(* CoDeSys 2.3.8.1 project: coconuts.pro *)
(* Libraries: C:\Program Files (x86)\Common Files\CAA-Targets\3S\Lib_PLCWinNT\SysLibTime.lib 23.9.04 10:11:36, STANDARD.LIB 4.10.05 11:14:46, IECSFC.LIB 13.4.06 15:51:28, Util.lib 1.6.07 09:40:58, ANALYZATION.LIB 5.10.99 09:05:06, C:\Program Files (x86)\Common Files\CAA-Targets\3S\Lib_PLCWinNT\SysLibFile.lib 23.9.04 10:11:36 *)

(* PLC configuration (modules and I/O channels)
Discrete input 6 bit [ID100] node 0, in %IB0 out %QB0 {Filtrationtime = 10; Filtrationtime = 10; Filtrationtime = 10; Filtrationtime = 10; Filtrationtime = 10; Filtrationtime = 10; Visibility = No; PinCount = 6; WatchDogPeriod = 1000; PollPeriod = 1}
  SW1 AT %IX0.0 [BitInput]
  SW2 AT %IX0.1 [BitInput]
  SW3 AT %IX0.2 [BitInput]
  SW4 AT %IX0.3 [BitInput] kitchen
  SW5 AT %IX0.4 [BitInput]
  SW6 AT %IX0.5 [BitInput] entrance
R1 AT %QX1.0 [BitOutput] water boiler
_R2 AT %QX1.1 [BitOutput]
_R3 AT %QX1.2 [BitOutput] entrance
R4 AT %QX1.3 [BitOutput] electro boiler
Special output [ID104] node 2, in %IB2 out %QB2 {Visibility = No; PinCount = 1}
  BEEPER AT %QX2.0 [BitOutput] Special output
Unifed signal sensor [ID700] node 3, in %IB3 out %QB3 {Type_of_sensor700 = U0_1; measure_interval = 1; ainlow = 0; ainhigh = 30; first_cor_point = 0; first_delta = 0; second_cor_point = 0; second_delta = 0; third_cor_point = 0; third_delta = 0; Visibility = No}
  AT %ID3.0 [FloatInput] Value
  AT %IW3.1 [WordInput] Circular time
  Analog Input [ID107] node 0, in %IB3.0 out %QB3.0
Unifed signal sensor [ID700] node 4, in %IB4 out %QB4 {Type_of_sensor700 = U0_1; measure_interval = 0.5; ainlow = 0; ainhigh = 20; first_cor_point = 0; first_delta = 0; second_cor_point = 0; second_delta = 0; third_cor_point = 0; third_delta = 0; Visibility = No}
  AT %ID4.0 [FloatInput] Value
  AT %IW4.1 [WordInput] Circular time
  Analog Input [ID107] node 0, in %IB4.0 out %QB4.0
Unifed signal sensor [ID700] node 5, in %IB5 out %QB5 {Type_of_sensor700 = U0_1; measure_interval = 0.5; ainlow = 0; ainhigh = 20; first_cor_point = 0; first_delta = 0; second_cor_point = 0; second_delta = 0; third_cor_point = 0; third_delta = 0; Visibility = No}
  AT %ID5.0 [FloatInput] Value
  AT %IW5.1 [WordInput] Circular time
  Analog Input [ID107] node 0, in %IB5.0 out %QB5.0
Unifed signal sensor [ID700] node 6, in %IB6 out %QB6 {Type_of_sensor700 = U0_1; measure_interval = 0.5; ainlow = 0; ainhigh = 20; first_cor_point = 0; first_delta = 0; second_cor_point = 0; second_delta = 0; third_cor_point = 0; third_delta = 0; Visibility = No}
  AT %ID6.0 [FloatInput] Value
  AT %IW6.1 [WordInput] Circular time
  Analog Input [ID107] node 0, in %IB6.0 out %QB6.0
Analog output [ID106] node 7, in %IB7 out %QB7 {DAC_Type = Voltage 0-10 B; Analog_offset_correction = 0; Analog_full_range_correction = 0; SafeValueFloat = 0; Visibility = No}
  AT %QD7.0 [FloatOutput] Value
Analog output [ID106] node 8, in %IB8 out %QB8 {DAC_Type = Voltage 0-10 B; Analog_offset_correction = 0; Analog_full_range_correction = 0; SafeValueFloat = 0; Visibility = No}
  AT %QD8.0 [FloatOutput] Value
ModBus (Master) [MODBUS_MASTER_ID450] node 9, in %IB9 out %QB9 {Visibility = No}
  MODBUS_LAST_ADDR AT %QD9.0 [DWordOutput] Last address
  MODBUS_LAST_ERROR AT %QW9.1 [WordOutput] Last error
  RS-485-1 [COM1_USART] node 0, in %IB9.0 out %QB9.0 {CommunicationSpeed = 9600; Parity = NO PARITY CHECK; BitLength = 8 bits; StopLength = One stop bit; InterfaceType = RS485; FrameOriented = RTU; Timeout = 0; Visibility = No}
  Universal Modbus device [ID2000] node 1, in %IB9.1 out %QB9.1 {ModuleIP = 10:0:0:223; ServiceTimeout = 150; TCPport = 502; NetMode = Serial; ModuleSlaveAddress = 3; RequestType = By poll time; PeriodOfService = 5000; Visibility = Yes; RepeatCounter = 0; ByteSequence = Trace_mode}
    AT %QB9.1.0 [ComChannel] Command (0xff - Start)
temp8 AT %IW9.1.0.0 [WordInput]
temp7 AT %IW9.1.1.0 [WordInput]
temp6 AT %IW9.1.2.0 [WordInput]
temp5 AT %IW9.1.3.0 [WordInput] 2f bedroom
temp4 AT %IW9.1.4.0 [WordInput] bath warm floor
temp3 AT %IW9.1.5.0 [WordInput] coolant
temp2 AT %IW9.1.6.0 [WordInput] living room
temp1 AT %IW9.1.7.0 [WordInput] boiler
Universal Modbus device [ID2000] node 2, in %IB9.2 out %QB9.2 {ModuleIP = 10:0:0:223; ServiceTimeout = 150; TCPport = 502; NetMode = Serial; ModuleSlaveAddress = 7; RequestType = By poll time; PeriodOfService = 5000; Visibility = Yes; RepeatCounter = 0; ByteSequence = Trace_mode}
  AT %QB9.2.0 [ComChannel] Command (0xff - Start)
temp78 AT %IW9.2.0.0 [WordInput] bedroom 2f
temp77 AT %IW9.2.1.0 [WordInput] hall
temp76 AT %IW9.2.2.0 [WordInput]
temp75 AT %IW9.2.3.0 [WordInput]
temp74 AT %IW9.2.4.0 [WordInput]
temp73 AT %IW9.2.5.0 [WordInput]
temp72 AT %IW9.2.6.0 [WordInput]
temp71 AT %IW9.2.7.0 [WordInput]
Universal Modbus device [ID2000] node 3, in %IB9.3 out %QB9.3 {ModuleIP = 10:0:0:223; ServiceTimeout = 150; TCPport = 502; NetMode = Serial; ModuleSlaveAddress = 2; RequestType = By poll time; PeriodOfService = 100; Visibility = Yes; RepeatCounter = 0; ByteSequence = Trace_mode}
  AT %QB9.3.0 [ComChannel] Command (0xff - Start)
AT %QB9.3.0.0 [ByteOutput]
Universal Modbus device [ID2000] node 4, in %IB9.4 out %QB9.4 {ModuleIP = 10:0:0:223; ServiceTimeout = 150; TCPport = 502; NetMode = Serial; ModuleSlaveAddress = 6; RequestType = By poll time; PeriodOfService = 100; Visibility = No; RepeatCounter = 0; ByteSequence = Trace_mode}
  AT %QB9.4.0 [ComChannel] Command (0xff - Start)
  8 bit input module [ID2001] node 0, in %IB9.4.0 out %QB9.4.0 {ModbusAddress = 0; Command_read_byte = Read inputs status  (0x02); Visibility = No}
    AT %IB9.4.0.0 [ByteInput]
AT %QB9.4.1.0 [ByteOutput]
AT %QB9.5.0 [ComChannel] Command (0xff - Start)
AT %QB9.5.0.0 [ByteOutput]
AT %IB9.5.1.0 [ByteInput]
Universal Modbus device [ID2000] node 6, in %IB9.6 out %QB9.6 {ModuleIP = 10:0:0:223; ServiceTimeout = 150; TCPport = 502; NetMode = Serial; ModuleSlaveAddress = 11; RequestType = By poll time; PeriodOfService = 20; Visibility = No; RepeatCounter = 0; ByteSequence = Trace_mode}
  AT %QB9.6.0 [ComChannel] Command (0xff - Start)
current AT %ID9.6.0.0 [FloatInput]
power AT %ID9.6.1.0 [FloatInput]
voltage AT %ID9.6.2.0 [FloatInput]
total_energy AT %ID9.6.3.0 [FloatInput]
Modbus [MODBUS_ID302] node 0, in %IB10.0 out %QB10.0
  TCP [TCP_ID221] node 0, in %IB10.0.0 out %QB10.0.0 {RemotePort = 502; Visibility = No}
REG0_LIGHTS16 AT %QW10.1.0 [WordOutput] reg0
REG1_PLC_FLAGS AT %QW10.2.0 [WordOutput] reg1
REG2_BOILERS AT %QW10.3.0 [WordOutput] reg2
REG3_PUMPS AT %QW10.4.0 [WordOutput] reg3
REG4_BATH_FAN_MODE AT %QW10.5.0 [WordOutput] reg4
REG5 AT %QW10.6.0 [WordOutput] reg5
REG6_LIVING_ROOM_TERMOSTAT_DESIRED AT %QW10.7.0 [WordOutput] reg6
REG7_HALL_TERMOSTAT_DESIRED AT %QW10.8.0 [WordOutput] reg7
REG8_2F_BEDROOM_TERMOSTAT_DESIRED AT %QW10.9.0 [WordOutput] reg8
REG9 AT %QW10.10.0 [WordOutput] reg9
REG10_TEMP1 AT %QW10.11.0 [WordOutput] reg10
REG11_TEMP2 AT %QW10.12.0 [WordOutput] reg11
REG12_TEMP3 AT %QW10.13.0 [WordOutput] reg12
REG13_TEMP4 AT %QW10.14.0 [WordOutput] reg13
REG14_TEMP5 AT %QW10.15.0 [WordOutput] reg14
REG15_TEMP6 AT %QW10.16.0 [WordOutput] reg15
REG16_TEMP7 AT %QW10.17.0 [WordOutput] reg16
REG17_TEMP8 AT %QW10.18.0 [WordOutput] reg17
REG18 AT %QW10.19.0 [WordOutput] reg18
REG19 AT %QW10.20.0 [WordOutput] reg19
REG20 AT %QW10.21.0 [WordOutput] reg20
REG21_POWER AT %QW10.22.0 [WordOutput]
REG22_VOLTAGE AT %QW10.23.0 [WordOutput]
REG23_TOTAL_ENERGY AT %QW10.24.0 [WordOutput]
REG24_TIME AT %QW10.25.0 [WordOutput]
ID4002 byteIB
%QB
%MB
%MREG25_MODBUS_ERRORS AT %QW10.26.0 [WordOutput]
REG26_BOILER_DESIRED_TEMP AT %QW10.27.0 [WordOutput]
REG27_BOILER_CUR_TEMP AT %QW10.28.0 [WordOutput]
REG28_BOILER_MODE AT %QW10.29.0 [WordOutput]
REG29_TEMP71 AT %QW10.30.0 [WordOutput]
REG30_TEMP72 AT %QW10.31.0 [WordOutput]
REG31_TEMP73 AT %QW10.32.0 [WordOutput]
REG32_TEMP74 AT %QW10.33.0 [WordOutput]
REG33_TEMP75 AT %QW10.34.0 [WordOutput]
REG34_TEMP76 AT %QW10.35.0 [WordOutput]
REG35_TEMP77 AT %QW10.36.0 [WordOutput]
REG36_TEMP78 AT %QW10.37.0 [WordOutput]
*)

(* Global variable list: Global_Variables *)
VAR_GLOBAL
	RO_POWER_NIGHT_MODE: BOOL;
	RO_POWER_SAFE_MODE:BOOL;

	WATER_BOILER_STATE:BOOL;
	RO_WATER_BOILER_VALVE_STATE:BOOL;

	RO_WARM_FLOOR_PUMP_STATE:BOOL;

	RO_LIVINGROOM_TERMOSTAT_STATE:BOOL;
	RO_BEDROOM_2F_TERMOSTAT_STATE:BOOL;

	RO_BEDROOM_2F_VALVE_STATE:BOOL;
	RO_HALL_VALVE_STATE:BOOL;

	TOWEL_HEATER_SW:switch;
	BATH_LIGHT_SW:switch;

	RO_BATH_FAN_STATE:BOOL;
END_VAR

VAR_GLOBAL CONSTANT
	MIN_COOLANT_TEMP: WORD := 300;
	MAX_COOLANT_TEMP: WORD := 600;
END_VAR

(* POU PLC_PRG, CFC *)
PROGRAM PLC_PRG
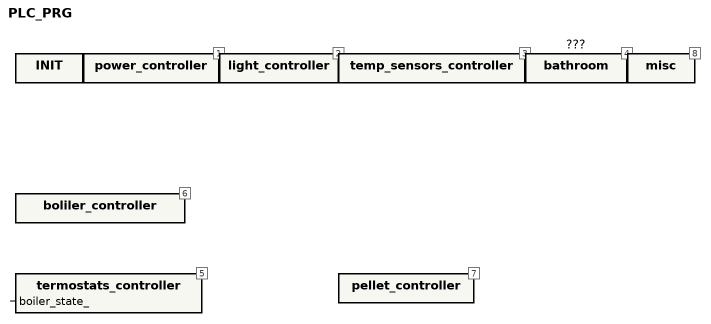
_CFC_ (* Continuous Function Chart, elements in execution order *)
#0 INIT()
#1 power_controller()
#2 light_controller()
#3 temp_sensors_controller()
#4 ???:bathroom()
#5 termostats_controller(boiler_state_: -)
#6 boliler_controller()
#7 pellet_controller()
#8 misc()
_END_CFC_
END_PROGRAM

(* POU INIT, ST *)
PROGRAM INIT
VAR
	initialized:BOOL := FALSE;
END_VAR
IF NOT initialized THEN
	initialized := TRUE;
	REG28_BOILER_MODE := 3;
	REG26_BOILER_DESIRED_TEMP := 450;
	REG6_LIVING_ROOM_TERMOSTAT_DESIRED := 225;
	REG8_2F_BEDROOM_TERMOSTAT_DESIRED := 225;
	REG7_HALL_TERMOSTAT_DESIRED := 225;

	R1 := FALSE;
	R4 := FALSE;

	RO_POWER_NIGHT_MODE:=FALSE;
	RO_POWER_SAFE_MODE:=FALSE;

	REG4_BATH_FAN_MODE := 1;
END_IF
END_PROGRAM

(* POU power_controller, ST *)
PROGRAM power_controller
VAR
	T : CurTimeEx;
	cur_date: SystemTimeDate;
	cur_time: SysTime64;

	timer: TON;
	energy_monitor_offline: BOOL := FALSE;

	FLAGS:ARRAY[0..15] OF BYTE;
	I: BYTE;

	BLINKER:BLINK;
	OVERLOAD_WARNING: BOOL := FALSE;
END_VAR
cur_date.dwLowMSecs := 0;
cur_date.dwHighMsec := 0;
cur_date.Milliseconds := 0;
cur_date.Minute := 0;
cur_date.Second := 0;
cur_date.Hour := 0;
cur_date.Day := 0;
cur_date.Year := 0;
cur_date.Month := 0;
cur_date.DayOfWeek := 0;

cur_time.ulHigh := 0;
cur_time.ulLow := 0;

T(SystemTime:=cur_time , TimeDate:=cur_date );

REG23_TOTAL_ENERGY := REAL_TO_WORD(total_energy);
REG24_TIME := SHL(UINT_TO_WORD(cur_date.Hour),8) OR UINT_TO_WORD(cur_date.Minute);

(* process flags *)
FOR I:=0 TO 15 DO
	FLAGS[I] :=BOOL_TO_BYTE( EXTRACT(REG1_PLC_FLAGS, i));
END_FOR

(* night-mode *)
IF  cur_date.Hour = 23 AND cur_date.Minute = 0 AND cur_date.Second = 0 THEN
	FLAGS[0] := 1;
ELSIF cur_date.Hour = 7 AND cur_date.Minute = 0 AND cur_date.Second = 0 THEN
	FLAGS[0] := 0;
END_IF

IF MODBUS_LAST_ADDR = 11 AND MODBUS_LAST_ERROR = 81 THEN
	energy_monitor_offline := TRUE;
ELSIF  MODBUS_LAST_ADDR = 11 AND MODBUS_LAST_ERROR = 0 THEN
	energy_monitor_offline := FALSE;
END_IF;

timer(IN:=energy_monitor_offline , PT:= T#10s , Q=> , ET=> );
FLAGS[1] := BOOL_TO_BYTE( BYTE_TO_BOOL(FLAGS[1]) OR timer.Q);
IF timer.Q THEN
	REG21_POWER := 0;
	REG22_VOLTAGE := 0;
ELSE
	REG21_POWER := REAL_TO_WORD(power);
	REG22_VOLTAGE := REAL_TO_WORD(voltage);
END_IF

RO_POWER_NIGHT_MODE := BYTE_TO_BOOL(FLAGS[0]);
RO_POWER_SAFE_MODE :=  BYTE_TO_BOOL(FLAGS[1]);

FOR I:=0 TO 15 DO
	REG1_PLC_FLAGS := DWORD_TO_WORD( PUTBIT(REG1_PLC_FLAGS, i, BYTE_TO_BOOL(FLAGS[I])));
END_FOR

(* sound warning *)
OVERLOAD_WARNING := REG21_POWER > 5500; (*OR RO_POWER_SAFE_MODE;*)
BLINKER(ENABLE:=OVERLOAD_WARNING, TIMELOW:=t#5s , TIMEHIGH:=t#300ms , OUT=> );
BEEPER := BLINKER.OUT AND OVERLOAD_WARNING;
END_PROGRAM

(* POU light_controller, ST *)
PROGRAM light_controller
VAR
	S0: switch;
	S1:switch;
	S2:switch;
	S3:switch;
	S4:switch;
	S6:switch;
	S7:switch;
	S8:switch;
	T1:F_TRIG;
	S0_R_TRIG:R_TRIG;
	S0_F_TRIG:F_TRIG;

	LIGHTS:ARRAY[0..15] OF BYTE;
	I: BYTE;
END_VAR
FOR I:=0 TO 15 DO
	LIGHTS[I] :=BOOL_TO_BYTE( EXTRACT(REG0_LIGHTS16, i));
END_FOR;

(* living room *)
S0(	in:=sw5_1, set:= , reset:= , state:=ADR(LIGHTS[0]), out=>relay2);

(* kitchen lamps *)
S1(	in:=SW1, set:= , reset:= , state:=ADR(LIGHTS[1]), out=>relay3 );

(* entrance *)
S2(	in:=SW4, set:= , reset:= , 	state:=ADR(LIGHTS[2]), out=>relay1 );

(* bathroom *)
BATH_LIGHT_SW(in:=sw5_2, set:= , reset:= , state:=ADR(LIGHTS[3]),  timeout := T#2h, out=>relay6_6 );

(* living room 2 *)
S0_R_TRIG(CLK:= S0.out, Q=> ); (* detect S0 turning off*)
S0_F_TRIG(CLK:= S0.out, Q=> ); (* detect S0 turning onf*)
S8(	in:=, set:=S0_R_TRIG.Q, reset:=S0_F_TRIG.Q, state:=ADR(LIGHTS[4]), out=>relay4);

(* 2f bedroom *)
S3(	in:=sw6_2, set:=, reset:= , state:=ADR(LIGHTS[5]), out=> relay6_1);

(* towel heater *)
TOWEL_HEATER_SW(in:=, set:=, reset:= , state:=ADR(LIGHTS[6]), timeout := T#6h, out=> );

(* 2f hall *)
S4(	in:=sw6_1, set:=, reset:= , state:=ADR(LIGHTS[7]), out=> relay6_4);

(* kitchen *)
S6(	in:=SW3, set:= , reset:= , 	state:=ADR(LIGHTS[9]), out=>relay8 );

(* stairs light  *)
S7(	in:=SW2, set:=, reset:= , state:=ADR(LIGHTS[10]),  timeout := T#10m, out=> relay6_5);
T1(CLK:=BATH_LIGHT_SW.out , Q=>S7.set );

(*REG0_LIGHTS16 := 0;*)
FOR I:=0 TO 15 DO
	REG0_LIGHTS16 := DWORD_TO_WORD( PUTBIT(REG0_LIGHTS16, i, BYTE_TO_BOOL(LIGHTS[I])));
END_FOR;
END_PROGRAM

(* POU switch, ST *)
FUNCTION_BLOCK switch
VAR_INPUT
	in:BOOL;
	set:BOOL;
	reset:BOOL;
	state: POINTER TO BOOL;
	timeout: TIME := T#6h;
END_VAR

VAR_OUTPUT
	out: BOOL;
END_VAR

VAR
	prev : BOOL := FALSE;
	timer:TON;
END_VAR
IF in =TRUE AND prev = FALSE THEN
	state^ := NOT state^;
END_IF
prev := in;

IF set THEN
	state^ := TRUE;
ELSIF reset THEN
	state^ := FALSE;
END_IF

out := state^;

timer(IN:=out AND NOT in , PT:=timeout, Q=> reset, ET=> );
END_FUNCTION_BLOCK

(* POU Temp/temp_sensors_controller, ST *)
PROGRAM temp_sensors_controller
VAR
END_VAR
REG10_TEMP1 := validate_temp(temp1, REG10_TEMP1);
REG11_TEMP2 := validate_temp(temp2, REG11_TEMP2);
REG12_TEMP3 := validate_temp(temp3, REG12_TEMP3);
REG13_TEMP4 := validate_temp(temp4, REG13_TEMP4);
REG14_TEMP5 := validate_temp(temp5, REG14_TEMP5);
REG15_TEMP6 := validate_temp(temp6, REG15_TEMP6);
REG16_TEMP7 := validate_temp(temp7, REG16_TEMP7);
REG17_TEMP8 := validate_temp(temp8, REG17_TEMP8);

REG29_TEMP71 := validate_temp(temp71, REG29_TEMP71);
REG30_TEMP72 := validate_temp(temp72, REG30_TEMP72);
REG31_TEMP73 := validate_temp(temp73, REG31_TEMP73);
REG32_TEMP74 := validate_temp(temp74, REG32_TEMP74);
REG33_TEMP75 := validate_temp(temp75, REG33_TEMP75);
REG34_TEMP76 := validate_temp(temp76, REG34_TEMP76);
REG35_TEMP77 := validate_temp(temp77, REG35_TEMP77);
REG36_TEMP78 := validate_temp(temp78, REG36_TEMP78);
END_PROGRAM

(* POU Temp/validate_temp, ST *)
FUNCTION validate_temp : WORD
VAR_INPUT
	in_temp: WORD;
	def_temp: WORD;
END_VAR
IF in_temp < 1 OR in_temp > 800 THEN
	validate_temp := def_temp;
ELSE
	validate_temp := in_temp;
END_IF
END_FUNCTION

(* POU bathroom, ST *)
PROGRAM bathroom
VAR
	fan_on: TON;
	fan_off: TOF;
	towel_heater: TON;
	towel_pwm: BLINK;
	fan_need:BOOL;
	fan_state:BOOL;
END_VAR
fan_on(IN:=BATH_LIGHT_SW.out,
		 PT:= T#1m,
		 Q=> ,
		 ET=> );

fan_off(IN:=fan_on.Q ,
		 PT:= T#10m,
		 Q=>fan_need ,
		 ET=> );


towel_heater(IN:=BATH_LIGHT_SW.out, PT:=T#10m, Q=>TOWEL_HEATER_SW.set);
towel_pwm(ENABLE:=TOWEL_HEATER_SW.out , TIMELOW:=T#10m , TIMEHIGH:=t#1m , OUT=>);
relay7 := TOWEL_HEATER_SW.out AND NOT towel_pwm.OUT;


IF REG4_BATH_FAN_MODE = 0 THEN
	fan_state := FALSE;
	fan_on.IN := FALSE;
	fan_off.in := FALSE;

ELSIF REG4_BATH_FAN_MODE =1 THEN
	fan_state := fan_need;

ELSIF REG4_BATH_FAN_MODE =2 THEN
	fan_state := TRUE;
END_IF


relay6_8 := fan_state;
RO_BATH_FAN_STATE := fan_state;
END_PROGRAM

(* POU Temp/termostats_controller, ST *)
PROGRAM termostats_controller
VAR
	living_room: termostat;
	bedroom2f: termostat;
	hall: termostat;
	unused: WORD;
END_VAR

VAR_INPUT
	boiler_state_: BOOL;
END_VAR
(*
	REG12_TEMP3 - coolant temp
      MIN_COOLANT_TEMP
*)

(* livingroom *)
living_room(	temp_in:= ADR(REG11_TEMP2) ,
				desired_temp_in:=ADR(REG6_LIVING_ROOM_TERMOSTAT_DESIRED),
				state_out := ADR(unused) ,
				delta:= 1,
				delay:= T#60m,
				out => );
RO_LIVINGROOM_TERMOSTAT_STATE := living_room.out;
RO_WARM_FLOOR_PUMP_STATE :=  living_room.out AND REG12_TEMP3 > (MIN_COOLANT_TEMP - 15);
relay5 := RO_WARM_FLOOR_PUMP_STATE;


(*bedroom2f *)
bedroom2f(	temp_in:= ADR(REG36_TEMP78) ,
				desired_temp_in:=ADR(REG8_2F_BEDROOM_TERMOSTAT_DESIRED),
				state_out := ADR(unused),
				delta:= 1,
				delay:= T#15m,
				out =>);
RO_BEDROOM_2F_TERMOSTAT_STATE := bedroom2f.out;
RO_BEDROOM_2F_VALVE_STATE := NOT bedroom2f.out AND REG12_TEMP3 > MIN_COOLANT_TEMP AND REG12_TEMP3 < MAX_COOLANT_TEMP;
relay5_5 := RO_BEDROOM_2F_VALVE_STATE;


(*hall *)
hall(temp_in:= ADR(REG35_TEMP77) ,
				desired_temp_in:=ADR(REG7_HALL_TERMOSTAT_DESIRED),
				state_out := ADR(unused),
				delta:= 1,
				delay:= T#15m,
				out =>);
RO_BEDROOM_2F_TERMOSTAT_STATE := bedroom2f.out;
RO_HALL_VALVE_STATE := NOT hall.out AND REG12_TEMP3 > MIN_COOLANT_TEMP AND REG12_TEMP3 < MAX_COOLANT_TEMP;
relay5_3 := RO_BEDROOM_2F_VALVE_STATE;
END_PROGRAM

(* POU Temp/termostat, ST *)
FUNCTION_BLOCK termostat
VAR_INPUT
	temp_in:POINTER TO WORD;
	desired_temp_in:POINTER TO WORD;
	state_out: POINTER TO BYTE;
	delta:BYTE;
	delay:TIME;
	set:BOOL;
	reset:BOOL;
END_VAR

VAR_OUTPUT
	out: BOOL;
END_VAR

VAR
	state: BOOL:=FALSE;
	timer_off: TON;
	timer_on: TON;
END_VAR
timer_off(PT := delay, IN := state);
timer_on(PT:=T#10s, IN :=  temp_in^ < desired_temp_in^ - delta);

IF temp_in^ > desired_temp_in^ + delta AND timer_off.Q THEN
	state := FALSE;
ELSIF timer_on.Q THEN
	state := TRUE;
END_IF

IF set THEN
	state := TRUE;
ELSIF reset THEN
	state := FALSE;
END_IF

state_out^ := BOOL_TO_BYTE(state);
out := state;
END_FUNCTION_BLOCK

(* POU Temp/boliler_controller, ST *)
PROGRAM boliler_controller

VAR
	unused: WORD := 0;
	P:overload_control;
	boiler_need: BOOL;
	electro_mode: BOOL;
	pellet_mode:BOOL;
	timer: TON;
END_VAR
(*
	REG10_TEMP1 - boiler raw  temp
	REG12_TEMP3 - coolant temp
	REG26_BOILER_DESIRED_TEMP
	REG27_BOILER_CUR_TEMP
      MIN_COOLANT_TEMP
	REG28_BOILER_MODE
*)

(* trainsitions *)
IF RO_POWER_SAFE_MODE THEN
	REG28_BOILER_MODE := 3;
END_IF

REG27_BOILER_CUR_TEMP := REG10_TEMP1;

IF REG27_BOILER_CUR_TEMP < REG26_BOILER_DESIRED_TEMP - 10 THEN
	boiler_need := TRUE;
ELSIF REG27_BOILER_CUR_TEMP > REG26_BOILER_DESIRED_TEMP + 10 THEN
	boiler_need := FALSE;
END_IF

(* off *)
IF REG28_BOILER_MODE = 0 THEN
	electro_mode := FALSE;
	pellet_mode := FALSE;

(* auto *)
ELSIF REG28_BOILER_MODE = 1 THEN
	IF REG12_TEMP3 > REG27_BOILER_CUR_TEMP AND REG12_TEMP3 > MIN_COOLANT_TEMP THEN
		pellet_mode := TRUE;
		electro_mode := FALSE;
	ELSE
		pellet_mode := FALSE;
		electro_mode := boiler_need;
	END_IF

(* electro *)
ELSIF REG28_BOILER_MODE = 2 THEN
	electro_mode := boiler_need;
	pellet_mode := FALSE;

(* pellet *)
ELSIF REG28_BOILER_MODE = 3 THEN
	pellet_mode := TRUE;
	electro_mode := FALSE;

(* turbo *)
ELSIF REG28_BOILER_MODE = 4 THEN
	pellet_mode := REG12_TEMP3 > REG27_BOILER_CUR_TEMP AND REG12_TEMP3 > MIN_COOLANT_TEMP;
	electro_mode := boiler_need;

END_IF

timer(IN:=NOT timer.Q , PT:= T#20m , Q=> , ET=> );

P(	in:= electro_mode,
	cur_power := REAL_TO_WORD(power),
	load_power := 2200,
	hi_limit_power := 4000,
	low_limit_power := 1000,
	cooldown := T#1m,
	reset := timer.Q,
	out => WATER_BOILER_STATE);


R1 := WATER_BOILER_STATE;
RO_WATER_BOILER_VALVE_STATE := pellet_mode;
relay5_1 := pellet_mode;
END_PROGRAM

(* POU overload_control, ST *)
FUNCTION_BLOCK overload_control
VAR_INPUT
	in: BOOL;
	cur_power: WORD;
	load_power: WORD;
	hi_limit_power : INT;
	low_limit_power : INT;
	cooldown: TIME;
	reset: BOOL;
END_VAR

VAR_OUTPUT
	out : BOOL;
END_VAR

VAR
	state: BOOL := FALSE;
	timer_on : TON;
	power_corrector : REAL;
	max_limit: INT;
END_VAR
power_corrector := voltage / 220;
max_limit :=0;

IF out = FALSE  THEN
	max_limit := REAL_TO_INT(cur_power + power_corrector * load_power);
	state := cur_power < low_limit_power AND max_limit < hi_limit_power;

ELSE
	state :=  cur_power < hi_limit_power;

END_IF

timer_on(	IN:= state AND NOT reset,
			PT:= cooldown,
			Q=>,
			ET=> );

out := in AND timer_on.Q;
END_FUNCTION_BLOCK

(* POU Temp/pellet_controller, ST *)
PROGRAM pellet_controller

VAR
	P: overload_control;
	awake: TOF;
	electro_boiler_enabled: BOOL;
END_VAR
(*
R4 -- electro bolier control
sw5_3 -- pelletes electro mode
*)

awake(IN:=BATH_LIGHT_SW.out , PT:=T#2m , Q=> , ET=> );
electro_boiler_enabled := sw5_3 AND NOT RO_POWER_SAFE_MODE; (* AND NOT awake.q; *)

P(	in:= electro_boiler_enabled,
	cur_power:=REAL_TO_WORD(power),
	load_power:=4200,
	hi_limit_power:=5300,
	low_limit_power:=500,
	cooldown := T#50s,
	reset := FALSE,
	out => R4);
END_PROGRAM

(* POU misc, ST *)
PROGRAM misc
VAR
	boilers:ARRAY[0..15] OF BYTE;
	pumps:ARRAY[0..15] OF BYTE;
	I: BYTE;

	succes_packets: WORD := 0;
	failed_packets: WORD := 0;
END_VAR
boilers[0] := BOOL_TO_BYTE(FALSE);
boilers[1] := BOOL_TO_BYTE(FALSE);
boilers[2] := BOOL_TO_BYTE(WATER_BOILER_STATE);
boilers[3] := BOOL_TO_BYTE(RO_LIVINGROOM_TERMOSTAT_STATE);
boilers[4] := BOOL_TO_BYTE(RO_BEDROOM_2F_TERMOSTAT_STATE);

pumps[0] := BOOL_TO_BYTE(RO_WATER_BOILER_VALVE_STATE);
pumps[1] := BOOL_TO_BYTE(RO_WARM_FLOOR_PUMP_STATE);
pumps[2] := BOOL_TO_BYTE(RO_BEDROOM_2F_VALVE_STATE);
pumps[3] := BOOL_TO_BYTE(RO_HALL_VALVE_STATE);
pumps[4] := BOOL_TO_BYTE(FALSE);
pumps[5] := BOOL_TO_BYTE(FALSE);
pumps[6] := BOOL_TO_BYTE(RO_BATH_FAN_STATE);

FOR I:=0 TO 15 DO
	REG2_BOILERS := DWORD_TO_WORD( PUTBIT(REG2_BOILERS, i, BYTE_TO_BOOL(boilers[I])));
END_FOR;

FOR I:=0 TO 15 DO
	REG3_PUMPS := DWORD_TO_WORD( PUTBIT(REG3_PUMPS, i, BYTE_TO_BOOL(pumps[I])));
END_FOR;


(* modbus errors *)
IF succes_packets > 1000 THEN
	REG25_MODBUS_ERRORS := 100 * failed_packets / succes_packets;
	failed_packets := 0;
	succes_packets := 0;
END_IF;

IF MODBUS_LAST_ERROR <> 0 THEN
	failed_packets := failed_packets + 1;
ELSE
	succes_packets := succes_packets + 1;
END_IF;
END_PROGRAM
